(* PLC project PlcMain, Beckhoff Automation GmbH TwinCAT PLC Control 3.5.13.21 *)
(* stored: creationDateTime 2022-08-19T12:34:02.7808916, modificationDateTime 2022-08-19T12:34:02.7808916 *)

{attribute 'qualified_only'}
{attribute 'strict'}
TYPE StateCnv :
(
	Off,
	Reset,
	Power,
	Ready,
	Moving
);
END_TYPE
